Universal Robots PolyScope program: 02_Trajectory_02_round.urp

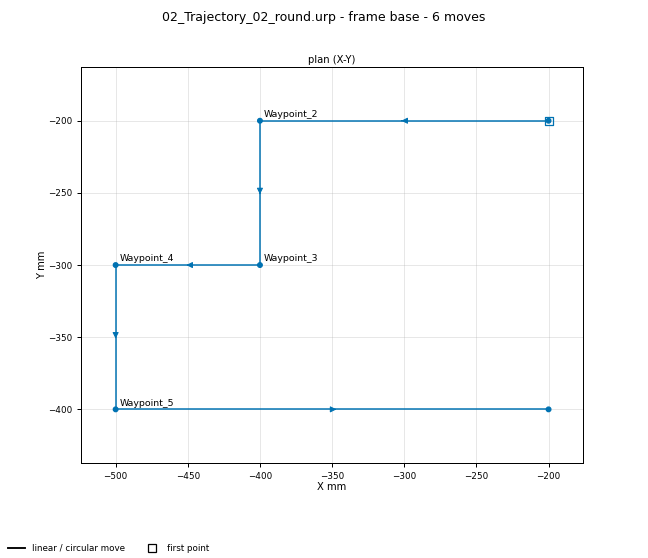
[picture p0: tool path of 02_Trajectory_02_round.urp in frame base, 6 of 6 moves have a stored position in this frame; points joined in program order, loops and branches not executed]
Program 02_Trajectory_02_round (installation=default directory=/home/ur/ursim-current/programs/Test_Programs createdIn=5.9.1.1031110 lastSavedIn=5.9.1.1031110 robotSerialNumber=20195599999)
Calibrated DH parameters: a=[0, -0.425, -0.3922, 0, 0, 0]; d=[0.1625, 0, 0, 0.1333, 0.0997, 0.0996]; alpha=[1.570796, 0, 0, 1.570796, -1.570796, 0]; deltaTheta=[0, 0, 0, 0, 0, 0]
Robot Program (runOnlyOnce=false)
  MoveL speed 250 mm/s, acceleration 1200 mm/s^2 (useActiveTCP=true) feature=Base
    Waypoint Waypoint_1: motionParameters(blendRadius=0.05); TCP in base x=-200 y=-200 z=200 mm, rx=0 ry=3.1416 rz=0 rad; joints [-106.882, -70.742, -151.59, -47.668, 90, -16.882] deg
    Waypoint Waypoint_2: motionParameters(blendRadius=0.05); TCP in base x=-400 y=-200 z=200 mm, rx=0 ry=3.1416 rz=0 rad; joints [-136.093, -97.679, -128.736, -43.585, 90, -46.093] deg
    Waypoint Waypoint_3: motionParameters(blendRadius=0.05); TCP in base x=-400 y=-300 z=200 mm, rx=0 ry=3.1416 rz=0 rad; joints [-127.668, -104.003, -120.574, -45.423, 90, -37.668] deg
    Waypoint Waypoint_4: motionParameters(blendRadius=0.048); TCP in base x=-500 y=-300 z=200 mm, rx=0 ry=3.1416 rz=0 rad; joints [-135.821, -113.339, -106.856, -49.805, 90, -45.821] deg
    Waypoint Waypoint_5: motionParameters(blendRadius=0.05); TCP in base x=-500 y=-400 z=200 mm, rx=0 ry=3.1416 rz=0 rad; joints [-129.324, -119.683, -96.607, -53.71, 90, -39.324] deg
    Waypoint Waypoint_6: motionParameters(blendRadius=0.05); TCP in base x=-200 y=-400 z=200 mm, rx=0 ry=3.1416 rz=0 rad; joints [-99.223, -97.679, -128.736, -43.585, 90, -9.223] deg
